INTERFACE IMover EXTENDS ZApplication.IUnit

END_INTERFACE

(* stored: Version 1.1.0.1
   Itf IMover: Id {c2c45bc0-60bf-4f71-a6a2-cfead6528737} *)
